// TIA Portal V20 export
// export: Created 2025-12-01T14:57:13.2854996Z, ExportSetting None, DisplayName Totally Integrated Automation Portal, DisplayVersion V20 Update 3, DisplayName TIA Portal Openness, DisplayVersion V20 Update 3, DisplayName TIA Portal Version Control Interface, DisplayVersion V20 Update 3, DisplayName STEP 7 Professional, DisplayVersion V20 Update 3, DisplayName STEP 7 Safety, DisplayVersion V20 Update 2, DisplayName WinCC Basic/Comfort/Advanced, DisplayVersion V20 Update 3, DisplayName WinCC Professional, DisplayVersion V20 Update 3, DisplayName WinCC Unified, DisplayVersion V20 Update 3
FUNCTION "FC882_FIFO_VisualizarErrores" : Void   // FC882, LAD
{ S7_Optimized_Access := 'FALSE' }
AUTHOR : ERRORES
NAME : 20160407
VERSION : 3.3
// stored: AutoNumber false, SetENOAutomatically false
   VAR_INPUT
      Actualiza : Bool;
   END_VAR
   VAR_IN_OUT
      CodigoError : UDInt;
      Tipo : UInt;
      Numero : UInt;
      Error : UInt;
   END_VAR
   VAR_TEMP
      MaxDispositivos : UInt;
      NumDispo : UInt;
      NumDispoAnterior : UInt;
      Indice : UInt;
   END_VAR
   VAR CONSTANT
      CTE_CCPIF_ErrorGrave : UInt := 0;   // CCPIF - Numero - Indice
      CTE_CBOX_ErrorGrave : UInt := 100;   // CBOX - Numero Maximo - Indice
      CTE_CCPIF_ErrorLeve : UInt := 101;   // CCPIF - Numero - Indice
      CTE_CBOX_ErrorLeve : UInt := 201;   // CBOX - Numero Maximo - Indice
      CTE_MESAS : UInt := 702;   // MESA - Numero Maximo - Indice
      CTE_MAQUINAS : UInt := 1203;   // MAQUINA - Numero Maximo - Indice
   END_VAR
BEGIN

NETWORK
TITLE = Inicializar Variables
///////////////////////////////////////////////////////////////////////////
///////////////////////////////////////////////////////////////////////////
///////////////////////////////////////////////////////////////////////////
// --- Inicializar Variables

      L     "CTE_MaxTodosDispositivos";  // Max que se puedeb configurar
      L     4;  // +4 dispositivos 0
      +I;
      L     1;
      -I;
      T     #MaxDispositivos;  // MaxDispositivos

      L     "DB861_FIFO_Errores".IndiceExtracion;
      T     #NumDispoAnterior;  // ispositivo Ultimo




NETWORK
TITLE = Comprobar si se visualiza siguiente ERROR
///////////////////////////////////////////////////////////////////////////
///////////////////////////////////////////////////////////////////////////
///////////////////////////////////////////////////////////////////////////
// --- Hay que actualizar Siguiente Error

      A     #Actualiza;
      JC    ActulizarVisualizacion;

      JU    FinalFuncion;



NETWORK
TITLE = DIstribucion dependiendo de Dispositivo
///////////////////////////////////////////////////////////////////////////
///////////////////////////////////////////////////////////////////////////
///////////////////////////////////////////////////////////////////////////
/// --- Distribucion dependiendo del tipo de Dispositivo
ActulizarVisualizacion:NOP   0;
      L     #NumDispoAnterior;
      L     1;
      +I;
      T     #NumDispo;  // Siguiente Dispositivo a Visualizar


/// --- Inicio de Bucle de Dispositivos
InicioBucle_Dispositivos:NOP   0;
      SET;  // CCPIF - Error Grave
      L     #NumDispo;
      L     #CTE_CCPIF_ErrorGrave;
      ==I;
      JC    CCPIF_Dispositivo_ErrorGrave;
      SET;  // CBOX - Error Grave
      L     #NumDispo;
      L     #CTE_CBOX_ErrorGrave;
      <=I;
      JC    CBOX_Dispositivo_ErrorGrave;


      SET;  // CCPIF - Error Leve
      L     #NumDispo;
      L     #CTE_CCPIF_ErrorLeve;
      ==I;
      JC    CCPIF_Dispositivo_ErrorLeve;
      SET;  // CBOX - Error Leve
      L     #NumDispo;
      L     #CTE_CBOX_ErrorLeve;
      <=I;
      JC    CBOX_Dispositivo_ErrorLeve;

      SET;  // MESA
      L     #NumDispo;
      L     #CTE_MESAS;
      <=I;
      JC    MESA_Dispositivo;

      SET;  // MAQUINA
      L     #NumDispo;
      L     #CTE_MAQUINAS;
      <=I;
      JC    MAQUINA_Dispositivo;

// No hay mas Dispositivos
//      SPA   NumeroMaximoDeDispositivos

///////////////////////////////////////////////////////////////////////////
///////////////////////////////////////////////////////////////////////////
///////////////////////////////////////////////////////////////////////////


///////////////////////////////////////////////////////////////////////////
///////////////////////////////////////////////////////////////////////////
///////////////////////////////////////////////////////////////////////////
/// Continuar el Bucle de Dispositivos
ContinuarBucle_Dispositivos:NOP   0;
      SET;  // La ha recorrido todos los Dispositivos ?
      L     #NumDispo;
      L     #NumDispoAnterior;
      ==I;
      JC    SinErrorDeDispositivos;

      SET;  // No hay Maximo de Dispositivos ?
      L     #NumDispo;
      L     #MaxDispositivos;
      >=I;
      JC    NumeroMaximoDeDispositivos;

      L     #NumDispo;
      L     1;
      +I;
      T     #NumDispo;  // Siguiente Dispositivo a Visualizar

      JU    InicioBucle_Dispositivos;


///////////////////////////////////////////////////////////////////////////
///////////////////////////////////////////////////////////////////////////
///////////////////////////////////////////////////////////////////////////
// --- Se ha recorrido todo el Array de Errores
NumeroMaximoDeDispositivos:NOP   0;
      L     0;
      T     #NumDispo;  // Empieza de Nuevo
      JU    InicioBucle_Dispositivos;


///////////////////////////////////////////////////////////////////////////
///////////////////////////////////////////////////////////////////////////
///////////////////////////////////////////////////////////////////////////
// --- No hay Errores a Visualizar
SinErrorDeDispositivos:NOP   0;
      L     0;
      T     #CodigoError;  // No hay Error
      T     #Tipo;
      T     #Numero;
      T     #Error;

      L     0;
      T     "DB861_FIFO_Errores".IndiceExtracion;
      JU    FinalFuncion;



NETWORK
TITLE = ---- Dispositivo >>> CCPIF -> ErrorGrave
///////////////////////////////////////////////////////////////////////////
///////////////////////////////////////////////////////////////////////////
///////////////////////////////////////////////////////////////////////////
/// --- Dispositivo >>> CCPIF - Error Grave
CCPIF_Dispositivo_ErrorGrave:NOP   0;
      L     0;  // - Dispositivo CCPIF
      T     #Indice;

      SET;  // Existe Error
      L     "DB861_FIFO_Errores".ArmariosGraves[#Indice];
      L     0;
      ==D;
      JC    ContinuarBucle_Dispositivos;


/// --- Nuevo Error a Visualizar
      L     50;  // Tipo >>> CCPIF
      T     #Tipo;

      L     "CTE_OffsetCCPIF";
      L     1;
      +I;
      T     #Numero;

      L     "DB861_FIFO_Errores".ArmariosGraves[#Indice];
      T     #Error;

      L     DINT#500000;
      L     #Numero;
      +D;
      L     DINT#1000;
      *D;
      L     #Error;
      +D;
      T     #CodigoError;

      L     #NumDispo;
      T     "DB861_FIFO_Errores".IndiceExtracion;
      JU    FinalFuncion;



NETWORK
TITLE = ---- Dispositivo >>> CCPIF -> ErrorLeves
///////////////////////////////////////////////////////////////////////////
///////////////////////////////////////////////////////////////////////////
///////////////////////////////////////////////////////////////////////////
/// --- Dispositivo >>> CCPIF - Error Leve
CCPIF_Dispositivo_ErrorLeve:NOP   0;
      L     #NumDispo;  // - Dispositivo CCPIF
      L     #CTE_CCPIF_ErrorLeve;
      -I;
      T     #Indice;

      SET;  // Existe Error
      L     "DB861_FIFO_Errores".ArmariosLeves[#Indice];
      L     0;
      ==D;
      JC    ContinuarBucle_Dispositivos;


/// --- Nuevo Error a Visualizar
      L     50;  // Tipo >>> CCPIF
      T     #Tipo;

      L     "CTE_OffsetCCPIF";
      L     1;
      +I;
      T     #Numero;

      L     "DB861_FIFO_Errores".ArmariosLeves[#Indice];
      T     #Error;

      L     DINT#500000;
      L     #Numero;
      +D;
      L     DINT#1000;
      *D;
      L     #Error;
      +D;
      T     #CodigoError;

      L     #NumDispo;
      T     "DB861_FIFO_Errores".IndiceExtracion;
      JU    FinalFuncion;



NETWORK
TITLE = ---- Dispositivo >>> CBOX -> ErrorGrave
///////////////////////////////////////////////////////////////////////////
///////////////////////////////////////////////////////////////////////////
///////////////////////////////////////////////////////////////////////////
/// --- Dispositivo >>> CBOX - Error Grave
CBOX_Dispositivo_ErrorGrave:NOP   0;
      L     #NumDispo;  // - Dispositivo CBOX
      T     #Indice;

      SET;  // Existe Error
      L     "DB861_FIFO_Errores".ArmariosGraves[#Indice];
      L     0;
      ==D;
      JC    ContinuarBucle_Dispositivos;


/// --- Nuevo Error a Visualizar
      L     40;  // Tipo >>> CBOX
      T     #Tipo;

      L     "CTE_OffsetCCPIF";
      L     1;
      +I;
      L     100;
      *I;
      L     #Indice;
      +I;
      T     #Numero;

      L     "DB861_FIFO_Errores".ArmariosGraves[#Indice];
      T     #Error;

      L     DINT#400000;
      L     #Numero;
      +D;
      L     DINT#1000;
      *D;
      L     #Error;
      +D;
      T     #CodigoError;

      L     #NumDispo;
      T     "DB861_FIFO_Errores".IndiceExtracion;
      JU    FinalFuncion;



NETWORK
TITLE = ---- Dispositivo >>> CBOX -> ErrorLeves
///////////////////////////////////////////////////////////////////////////
///////////////////////////////////////////////////////////////////////////
///////////////////////////////////////////////////////////////////////////
CBOX_Dispositivo_ErrorLeve:NOP   0;
      L     #NumDispo;  // - Dispositivo CBOX
      L     #CTE_CCPIF_ErrorLeve;
      -I;
      T     #Indice;

      SET;  // Existe Error
      L     "DB861_FIFO_Errores".ArmariosLeves[#Indice];
      L     0;
      ==D;
      JC    ContinuarBucle_Dispositivos;


/// --- Nuevo Error a Visualizar
      L     40;  // Tipo >>> CBOX
      T     #Tipo;

      L     "CTE_OffsetCCPIF";
      L     1;
      +I;
      L     100;
      *I;
      L     #Indice;
      +I;
      T     #Numero;

      L     "DB861_FIFO_Errores".ArmariosLeves[#Indice];
      T     #Error;

      L     DINT#400000;
      L     #Numero;
      +D;
      L     DINT#1000;
      *D;
      L     #Error;
      +D;
      T     #CodigoError;

      L     #NumDispo;
      T     "DB861_FIFO_Errores".IndiceExtracion;
      JU    FinalFuncion;



NETWORK
TITLE = ---- Dispositivo >>> MESA
///////////////////////////////////////////////////////////////////////////
///////////////////////////////////////////////////////////////////////////
///////////////////////////////////////////////////////////////////////////
MESA_Dispositivo:NOP   0;
      L     #NumDispo;  // - Dispositivo MESA
      L     #CTE_CBOX_ErrorLeve;
      -I;
      L     1;
      -I;
      T     #Indice;

      SET;  // Existe Error
      L     "DB861_FIFO_Errores".Mesas[#Indice];
      L     0;
      ==D;
      JC    ContinuarBucle_Dispositivos;


/// --- Nuevo Error a Visualizar
      L     60;  // Tipo >>> MESA
      T     #Tipo;

      L     "CTE_OffsetMesa";
      L     #Indice;
      +D;
      T     #Numero;

      L     "DB861_FIFO_Errores".Mesas[#Indice];
      T     #Error;

      L     DINT#600000;
      L     #Numero;
      +D;
      L     DINT#1000;
      *D;
      L     #Error;
      +D;
      T     #CodigoError;

      L     #NumDispo;
      T     "DB861_FIFO_Errores".IndiceExtracion;
      JU    FinalFuncion;



NETWORK
TITLE = ---- Dispositivo >>> MAQUINA
///////////////////////////////////////////////////////////////////////////
///////////////////////////////////////////////////////////////////////////
///////////////////////////////////////////////////////////////////////////
MAQUINA_Dispositivo:NOP   0;
      L     #NumDispo;  // - Dispositivo MAQUINA
      L     #CTE_MESAS;
      -I;
      L     1;
      -I;
      T     #Indice;

      SET;  // Existe Error
      L     "DB861_FIFO_Errores".Maquinas[#Indice];
      L     0;
      ==D;
      JC    ContinuarBucle_Dispositivos;


/// --- Nuevo Error a Visualizar
      L     70;  // Tipo >>> MAQUINA
      T     #Tipo;

      L     "CTE_OffsetMesa";
      L     #Indice;
      +I;
      T     #Numero;

      L     "DB861_FIFO_Errores".Maquinas[#Indice];
      T     #Error;

      L     DINT#700000;
      L     #Numero;
      +D;
      L     DINT#1000;
      *D;
      L     #Error;
      +D;
      T     #CodigoError;

      L     #NumDispo;
      T     "DB861_FIFO_Errores".IndiceExtracion;
      JU    FinalFuncion;



NETWORK
TITLE = Final de la funcion
///////////////////////////////////////////////////////////////////////////
///////////////////////////////////////////////////////////////////////////
///////////////////////////////////////////////////////////////////////////
// --- Final de la funcion

FinalFuncion:NOP   0;

END_FUNCTION
